FUNCTION CTRL_IN
  (* Standard: 61499-1 *)
  (* Version 1.0, 2025-12-19, franz *)
  PACKAGE OSCAT::Basic::POUs::Engineering::Control;
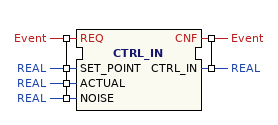
  EVENT_INPUT
    REQ WITH SET_POINT, ACTUAL, NOISE;
  END_EVENT
  EVENT_OUTPUT
    CNF WITH CTRL_IN;
  END_EVENT
  VAR_INPUT
    SET_POINT : REAL;
    ACTUAL : REAL;
    NOISE : REAL;
  END_VAR
  VAR_OUTPUT
    CTRL_IN : REAL;
  END_VAR
  BODY IN ST:
PACKAGE OSCAT::Basic::POUs::Engineering::Control;

FUNCTION CTRL_IN : REAL

VAR_INPUT
	SET_POINT : REAL;
	ACTUAL : REAL;
	NOISE : REAL;
END_VAR

(* calculate the process error DIFF *)
CTRL_IN := DEAD_ZONE(SET_POINT - ACTUAL, NOISE);

(* revision history hm 	2. jun. 2008 	rev 1.0 original version *)
END_FUNCTION
  END_BODY
END_FUNCTION
